FUNCTION_BLOCK FB_2_Skill_ROS2 EXTENDS FB_1_Skill
VAR_INPUT
// 	{attribute 'OPC.UA.DA.StructuredType':=1}
// 	{attribute 'OPC.UA.DA' := '1'}
// 	Control     : ST_SkillControl;
// 	{attribute 'OPC.UA.DA.StructuredType':=1}
// 	{attribute 'OPC.UA.DA' := '1'}
//     Status      : stExternalStatus;

//     Specific    : ST_RobotMoveSpecific;
	
END_VAR
VAR_OUTPUT
END_VAR
VAR
END_VAR

CYCLIC_ROS2();

ACTION CYCLIC_ROS2:
CYCLIC_SKILL();
END_ACTION

METHOD PROTECTED onActivate : eResult
VAR_INPUT
END_VAR

VAR
	eParentResult: eResult;
	myResult: ERESULT;
END_VAR

VAR //YOUR CODE
	succ : BOOL;
END_VAR
eParentResult := SUPER^.onActivate();
//--------------------------------------------------
myResult:=NONE;
// ----- YOUR CODE HERE (incl. Alarms) -------------

myResult:=NONE;

// ----- END YOUR CODE -----------------------------
//--------------------------------------------------
onActivate := CombineResults(eParentResult,myResult);
END_METHOD

METHOD PROTECTED onCleanup : eResult
VAR_INPUT
END_VAR

VAR
	eParentResult: eResult;
	myResult: ERESULT;
END_VAR

VAR //YOUR CODE
	succ : BOOL;
END_VAR
eParentResult := SUPER^.onCleanup();
//--------------------------------------------------
myResult:=NONE;
// ----- YOUR CODE HERE (incl. Alarms) -------------

myResult:=NONE;

// ----- END YOUR CODE -----------------------------
//--------------------------------------------------
onCleanup := CombineResults(eParentResult,myResult);
END_METHOD

METHOD PROTECTED onConfigure : eResult
VAR_INPUT
END_VAR

VAR
	eParentResult: eResult;
	myResult: ERESULT;
END_VAR

VAR //YOUR CODE
	succ : BOOL;
END_VAR
eParentResult := SUPER^.onConfigure();
//--------------------------------------------------
myResult:=NONE;
// ----- YOUR CODE HERE (incl. Alarms) -------------

myResult:=NONE;

// ----- END YOUR CODE -----------------------------
//--------------------------------------------------
onConfigure := CombineResults(eParentResult,myResult);
END_METHOD

METHOD PROTECTED onDeactivate : eResult
VAR_INPUT
END_VAR

VAR
	eParentResult: eResult;
	myResult: ERESULT;
END_VAR

VAR //YOUR CODE
	succ : BOOL;
END_VAR
eParentResult := SUPER^.onDeactivate();
//--------------------------------------------------
myResult:=NONE;
// ----- YOUR CODE HERE (incl. Alarms) -------------

myResult:=NONE;

// ----- END YOUR CODE -----------------------------
//--------------------------------------------------
onDeactivate := CombineResults(eParentResult,myResult);
END_METHOD

METHOD PROTECTED onError : eResult
VAR_INPUT
END_VAR

VAR
	eParentResult: eResult;
	myResult: ERESULT;
END_VAR

VAR //YOUR CODE
	succ : BOOL;
END_VAR
eParentResult := SUPER^.onError();
//--------------------------------------------------
myResult:=NONE;
// ----- YOUR CODE HERE (incl. Alarms) -------------

myResult:=NONE;

// ----- END YOUR CODE -----------------------------
//--------------------------------------------------
onError := CombineResults(eParentResult,myResult);
END_METHOD

METHOD PROTECTED onShutdown : eResult
VAR_INPUT
END_VAR

VAR
	eParentResult: eResult;
	myResult: ERESULT;
END_VAR

VAR //YOUR CODE
	succ : BOOL;
END_VAR
eParentResult := SUPER^.onShutdown();
//--------------------------------------------------
myResult:=NONE;
// ----- YOUR CODE HERE (incl. Alarms) -------------

myResult:=NONE;

// ----- END YOUR CODE -----------------------------
//--------------------------------------------------
onShutdown := CombineResults(eParentResult,myResult);
END_METHOD

END_FUNCTION_BLOCK

(* stored: Version 1.1.0.1, ProductVersion 3.1.4026.18
   POU FB_2_Skill_ROS2: Id {2e00d6a1-8d22-4bf8-a533-217a1a8bd953}, SpecialFunc None
   Folder StateControl: Id {a0d7267b-99f4-41f2-8af1-fa0fbdfbdb62}
   Action CYCLIC_ROS2: Id {e850367c-2480-40a1-a151-25b4245f1759}
   Method onActivate: Id {bc2d83b7-2512-4688-a8e1-54e2299564c4}
   Method onCleanup: Id {6fd91c29-8e32-488f-9ae6-151d92027456}
   Method onConfigure: Id {d115cc8e-7f1a-49b5-899a-a8343b56dd26}
   Method onDeactivate: Id {88519088-d0f4-44de-be30-f5617d391955}
   Method onError: Id {6f028444-e95e-464c-8fca-f4509fc4038a}
   Method onShutdown: Id {46466cbc-d126-42d4-a4a0-92feae79e9e1} *)
